TYPE csp_case_tr_accU_ls_width_enum :
(
	CSP_CASE_TR_ACCU_LS_WIDTH_STATUS_NOT_INITIALIZED 								:= 0,
	CSP_CASE_TR_ACCU_LS_WIDTH_STATUS_DISABLED 										:= 10,
	CSP_CASE_TR_ACCU_LS_WIDTH_STATUS_POSITION_CHECK									:= 20,
	CSP_CASE_TR_ACCU_LS_WIDTH_STATUS_ENABLE_REQUEST 								:= 30,
	CSP_CASE_TR_ACCU_LS_WIDTH_STATUS_ENABLED 										:= 40,
	CSP_CASE_TR_ACCU_LS_WIDTH_STATUS_GEAR_REQUEST									:= 50,
	CSP_CASE_TR_ACCU_LS_WIDTH_STATUS_GEARING										:= 60,
	CSP_CASE_TR_ACCU_LS_WIDTH_STATUS_GEARED											:= 70,
	CSP_CASE_TR_ACCU_LS_WIDTH_STATUS_MOVING											:= 80,
	CSP_CASE_TR_ACCU_LS_WIDTH_STATUS_DISENGAGE_REQUEST								:= 90,
	CSP_CASE_TR_ACCU_LS_WIDTH_STATUS_DISENGAGING									:= 100,
	CSP_CASE_TR_ACCU_LS_WIDTH_STATUS_STOP_REQUEST 									:= 110,
	CSP_CASE_TR_ACCU_LS_WIDTH_STATUS_DISABLE_REQUEST 								:= 120,
	CSP_CASE_TR_ACCU_LS_WIDTH_STATUS_DISABLING 										:= 130
) := CSP_CASE_TR_ACCU_LS_WIDTH_STATUS_NOT_INITIALIZED;
END_TYPE

(* stored: Version 1.1.0.1, ProductVersion 3.1.4024.3
   DUT csp_case_tr_accU_ls_width_enum: Id {2ed8870e-2933-4dfc-bdb6-96ccbc0daea9} *)
